ABB RobotStudio station: p3_robotstudio_2parte.rspag

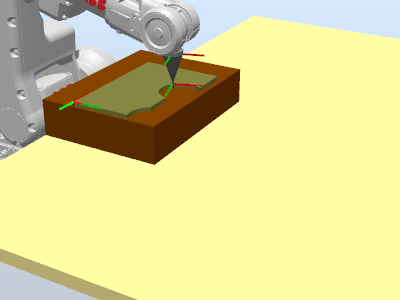
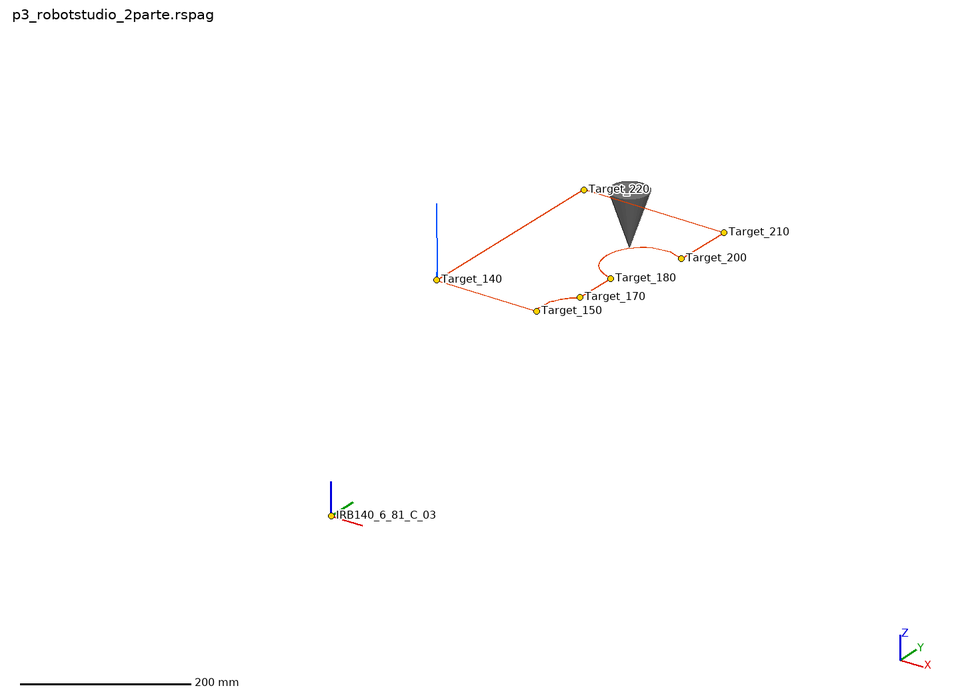
[picture v1: parts stored in the station drawn from their meshes, with robot base, taught points and paths (robot models come from the ABB library and are not in the file)]
--- station ---
Station p3_robotstudio_2parte (saved by RobotStudio 22.2.10013.1)
Controller Controlador1
  mechanical unit ROB_1: IRB140_6_81_C_03, 6 joints, base frame (0, 0, 0) mm
Layout (positions relative to the parent item):
  - printbed_hemisphere_hexagono [part, from P3_RobotStudio\hemisphere.rslib] at (471.3, 85, 364.75) mm, rotated rx 90 ry 0 rz 0 deg
  - Mesa de trabajo [part, from P3_RobotStudio\Mesa de trabajoDISA.rslib] at (1200, -600, -395) mm, rotated rx 0 ry 0 rz 90 deg
  - Pieza1 [part, from P3_RobotStudio\Pieza_ampliacion.rslib] at (500, 0, 200) mm, rotated rx 0 ry 0 rz 90 deg
  - trazador [smart component, from P3_RobotStudio\trazador.rslib] at (420.28, 9.26, 538.39) mm, rotated rx 179.65 ry 0.12 rz 18.57 deg
      connections:
        trazador.entrada_inyector -> TraceTCP.Enabled
        trazador.entrada_inyector -> ?.InputA
        ?.Output -> TraceTCP.Clear
    - TraceTCP [smart component, from Components\TraceTCP.rslib]
        properties: Robot=IRB140_6_81_C_03
  - IRB140_6_81_C_03 [mechanism, from Robots\IRB140_6_81_C_G_03.rslib] at (0, 0, 0) mm; joint values [0.023, -0.0385, 0.3276, -0.0067, 1.2818, 2.8424] (rad or m)
  - tool_laser [part] at (420.28, 9.26, 538.39) mm, rotated rx 179.65 ry 0.12 rz 18.57 deg, size 50 x 49.9 x 75 mm
  - tool_laser [mechanism] at (420.28, 9.26, 538.39) mm, rotated rx 179.65 ry 0.12 rz 18.57 deg
      TCP tool_laser at (0, 0, 75) mm
      links: Pieza_1
  - Curve_thing [part, from Training Objects\Curve_Thing.rslib] at (499.94, -199.87, 364.72) mm, rotated rx 0 ry 0.37 rz 89.92 deg
Attachment: trazador is attached to IRB140_6_81_C_03 / Link6
Attachment: tool_laser is attached to IRB140_6_81_C_03 / Link6
Attachment: tool_laser is attached to IRB140_6_81_C_03 / Link6
Station logic (signal -> signal, property => property):
  Controlador1.activar_mecanizado -> trazador.entrada_inyector

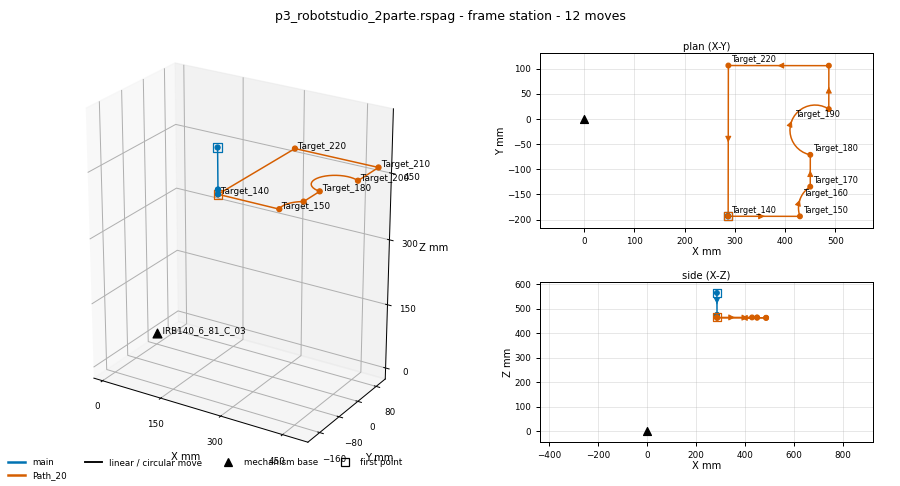
[picture p0: tool path of p3_robotstudio_2parte.rspag in frame station, 12 of 12 moves have a stored position in this frame; points joined in program order, loops and branches not executed]
--- Backups/Controlador1/RAPID/TASK1/PROGMOD/CalibData.mod ---
MODULE CalibData
    PERS tooldata tool_laser:=[TRUE,[[0,0,75],[1,0,0,0]],[1,[0,0,1],[1,0,0,0],0,0,0]];
    TASK PERS wobjdata Workobject:=[FALSE,TRUE,"",[[0,0,0],[1,0,0,0]],[[286.627001811,-193.490730871,464.561998296],[0.002682563,0.707605914,0.706600086,0.001729967]]];
    TASK PERS wobjdata wobj_mecanizado:=[FALSE,TRUE,"",[[0,0,0],[1,0,0,0]],[[286.627001811,-193.490730871,464.561998296],[0.002682563,0.707605914,0.706600086,0.001729967]]];
ENDMODULE

--- Backups/Controlador1/RAPID/TASK1/PROGMOD/MainModule.mod ---
MODULE MainModule
	PROC main()
        MoveJ Offs(Target_140,0,0,-100),v100,z100,tool_laser\WObj:=wobj_mecanizado;
        MoveL Offs(Target_140,0,0,-10),v30,fine,tool_laser\WObj:=wobj_mecanizado;
        MoveL Target_140,v5,fine,tool_laser\WObj:=wobj_mecanizado;
        Path_20;
        MoveL Offs(Target_140,0,0,-10),v30,fine,tool_laser\WObj:=wobj_mecanizado;
    ENDPROC
ENDMODULE

--- Backups/Controlador1/RAPID/TASK1/PROGMOD/Module1.mod ---
MODULE Module1

    CONST robtarget Target_140:=[[-0.001044518,0.001237331,-0.119945019],[0.707118807,0.00041804,-0.0039884,0.707083383],[0,0,0,0],[9E+09,9E+09,9E+09,9E+09,9E+09,9E+09]];
    CONST robtarget Target_150:=[[0.00386513,142.872007259,0.770403421],[0.707118807,0.00041804,-0.0039884,0.707083383],[0,0,0,0],[9E+09,9E+09,9E+09,9E+09,9E+09,9E+09]];
    CONST robtarget Target_160:=[[33.145326632,142.71973051,0.936803286],[0.986143735,0.0026539,-0.003006478,0.165844662],[0,0,0,0],[9E+09,9E+09,9E+09,9E+09,9E+09,9E+09]];
    CONST robtarget Target_170:=[[59.100802816,163.32684758,1.196283016],[0.875444758,0.001507495,-0.003716121,0.483301555],[0,0,0,0],[9E+09,9E+09,9E+09,9E+09,9E+09,9E+09]];
    CONST robtarget Target_180:=[[122.520192337,163.322672707,1.516495109],[0.999991959,0.003115824,-0.002524627,-0.000025048],[0,0,0,0],[9E+09,9E+09,9E+09,9E+09,9E+09,9E+09]];
    CONST robtarget Target_190:=[[190.312689625,126.331594958,1.628299126],[0.981718547,0.002578379,-0.003071491,0.190296119],[0,0,0,0],[9E+09,9E+09,9E+09,9E+09,9E+09,9E+09]];
    CONST robtarget Target_200:=[[213.534871513,199.983297206,2.204533414],[0.476705541,-0.000734056,-0.003942493,0.879053892],[0,0,0,0],[9E+09,9E+09,9E+09,9E+09,9E+09,9E+09]];
    CONST robtarget Target_210:=[[300.002003583,199.97760511,2.641116318],[0.999991959,0.003115824,-0.002524627,-0.000025048],[0,0,0,0],[9E+09,9E+09,9E+09,9E+09,9E+09,9E+09]];
    CONST robtarget Target_220:=[[299.995130863,-0.018511296,1.394771596],[0.707083383,0.0039884,0.00041804,-0.707118807],[0,0,0,0],[9E+09,9E+09,9E+09,9E+09,9E+09,9E+09]];
    CONST robtarget Target_230:=[[-0.001044518,0.001237331,-0.119945019],[0.000025048,-0.002524627,-0.003115824,0.999991959],[0,0,0,0],[9E+09,9E+09,9E+09,9E+09,9E+09,9E+09]];
    PROC Path_20()
        MoveL Target_140,v10,fine,tool_laser\WObj:=wobj_mecanizado;
        MoveL Target_150,v10,fine,tool_laser\WObj:=wobj_mecanizado;
        MoveC Target_160,Target_170,v10,fine,tool_laser\WObj:=wobj_mecanizado;
        MoveL Target_180,v10,fine,tool_laser\WObj:=wobj_mecanizado;
        MoveC Target_190,Target_200,v10,fine,tool_laser\WObj:=wobj_mecanizado;
        MoveL Target_210,v10,fine,tool_laser\WObj:=wobj_mecanizado;
        MoveL Target_220,v10,fine,tool_laser\WObj:=wobj_mecanizado;
        MoveL Target_230,v10,fine,tool_laser\WObj:=wobj_mecanizado;
    ENDPROC
ENDMODULE

--- Backups/Controlador1/SYSPAR/EIO.cfg ---
EIO:CFG_1.0:6:1::
#
EIO_SIGNAL:

      -Name "activar_mecanizado" -SignalType "DO" -Access "All"
